TYPE DUT_STRUCT_VARIABLES :
STRUCT
	sCellName			:STRING;
	sIpAddress			:STRING;
	sAmsNetId			:STRING;
	sOpcUaURL			:STRING;
	sUhfRfidOpcUaURL	:STRING;
	sHfRfidOpcUaURL		:STRING;
	sStation1			:STRING;
	sStation2			:STRING;
END_STRUCT
END_TYPE

(* stored: Version 1.1.0.1, ProductVersion 3.1.4024.6
   DUT DUT_STRUCT_VARIABLES: Id {75fee008-bd74-4965-a6e1-e2126a79bf49} *)
